FUNCTION_BLOCK FB_ReadParameterNC IMPLEMENTS I_ReadParameter
(*
    Read and refresh axis parameters
*)
VAR
    {attribute 'no_copy'}
    AxisRef : REFERENCE TO AXIS_REF;
// NC parameters that are exposed with pytmc pragmas
    {attribute 'pytmc' := '
        pv: PLC:AxisPar
        io: i
        field: DESC Axis configuration parameters in the numerical controller.
    '}
    stAxisParametersExposed : ST_AxisParameterSetExposed;

    // MC_ReadParameterSet Output
    fbMcReadParams: MC_ReadParameterSet;
    //{attribute 'hide'}
    stAxisParameters: ST_AxisParameterSet;
    bNcParamsReadInit   : BOOL;
    NCParamsTimer : TON;
    bAxisParametersInit : BOOL;
    tRefreshDelay: TIME := T#1S;
    bEnable : BOOL;
    bExecute : BOOL;
    bError				: BOOL;
    nErrorId			: UDINT:=0;
    sMessage : T_MAXSTRING;
    bDone : BOOL;
    bBusy    : BOOL;
END_VAR

PROPERTY Aborted : BOOL
GET
END_GET
END_PROPERTY

PROPERTY Active : BOOL
GET
END_GET
END_PROPERTY

PROPERTY AmsNetID : T_AmsNetId
GET
AmsNetID := THIS^.stAxisParameters.sAmsNetId;
END_GET
END_PROPERTY

PROPERTY AxisReadParamsInit : BOOL
GET
AxisReadParamsInit := bAxisParametersInit;
END_GET
END_PROPERTY

PROPERTY Busy : BOOL
GET
Busy := bBusy;
END_GET
END_PROPERTY

METHOD PUBLIC CallAfterInit
VAR_INPUT
    AxisRef : REFERENCE TO AXIS_REF;
END_VAR
THIS^.AxisRef REF= AxisRef;
END_METHOD

PROPERTY Done : BOOL
GET
Done := bDone;
END_GET
END_PROPERTY

PROPERTY EnInTargetTimeout : BOOL
GET
EnInTargetTimeout := THIS^.stAxisParameters.bEnablePEHTimeControl.0;
END_GET
END_PROPERTY

PROPERTY EnMaxSoftPosLimit : BOOL
GET
EnMaxSoftPosLimit := THIS^.stAxisParameters.bEncEnableSoftEndMaxControl.0;
END_GET
END_PROPERTY

PROPERTY EnMinSoftPosLimit : BOOL
GET
EnMinSoftPosLimit := THIS^.stAxisParameters.bEncEnableSoftEndMinControl.0;
END_GET
END_PROPERTY

PROPERTY EnPositionLagMonitoring : BOOL
GET
EnPositionLagMonitoring := THIS^.stAxisParameters.bCtrlEnablePosDiffControl.0;
END_GET
END_PROPERTY

PROPERTY EnPositionRangeMonitoring : BOOL
GET
END_GET
END_PROPERTY

PROPERTY EnScaleFactorInternal : LREAL
GET
EnScaleFactorInternal := THIS^.stAxisParameters.fEncScaleFactorInternal;
END_GET
END_PROPERTY

PROPERTY EnTargetPositionMonitoring : BOOL
GET
EnTargetPositionMonitoring := THIS^.stAxisParameters.bEnableTargetPosControl.0;
END_GET
END_PROPERTY

PROPERTY Error : BOOL
GET
Error := bError;
END_GET
END_PROPERTY

PROPERTY ErrorID : UDINT
GET
ErrorID := nErrorID;
END_GET
END_PROPERTY

//FB_Init is always available implicitly and it is used primarily for initialization.
//The return value is not evaluated. For a specific influence, you can also declare the
//methods explicitly and provide additional code there with the standard initialization
//code. You can evaluate the return value.
METHOD FB_Init: BOOL
VAR_INPUT
    bInitRetains: BOOL; // TRUE: the retain variables are initialized (reset warm / reset cold)
    bInCopyCode: BOOL;  // TRUE: the instance will be copied to the copy code afterward (online change)
    AxisRef : REFERENCE TO AXIS_REF;
END_VAR
THIS^.AxisRef REF= AxisRef;
END_METHOD

PROPERTY InTargetTimeout : LREAL
GET
InTargetTimeout := THIS^.stAxisParameters.fPEHControlTime;
END_GET
END_PROPERTY

PROPERTY MaxPosLagFilterTime : LREAL
GET
MaxPosLagFilterTime := THIS^.stAxisParameters.fCtrlPosDiffMaxTime;
END_GET
END_PROPERTY

PROPERTY MaxPosLagValue : LREAL
GET
MaxPosLagValue := THIS^.stAxisParameters.fCtrlPosDiffMax;
END_GET
END_PROPERTY

PROPERTY MaxSoftPosLimit : LREAL
GET
MaxSoftPosLimit := THIS^.stAxisParameters.fEncSoftEndMax;
END_GET
END_PROPERTY

PROPERTY Message : T_MAXSTRING
GET
Message := sMessage;
END_GET
END_PROPERTY

PROPERTY MinSoftPosLimit : LREAL
GET
MinSoftPosLimit := THIS^.stAxisParameters.fEncSoftEndMin;
END_GET
END_PROPERTY

PROPERTY Port : WORD
GET
Port := THIS^.stAxisParameters.nPort;
END_GET
END_PROPERTY

PROPERTY PositionRangeWindow : LREAL
GET
END_GET
END_PROPERTY

METHOD ReadParameters
VAR_INPUT
    Enable: BOOL;
    RefreshDelay: TIME;
END_VAR
THIS^.bEnable:= Enable;
THIS^.tRefreshDelay:= RefreshDelay;
END_METHOD

PROPERTY RefVeloSearch : LREAL
GET
RefVeloSearch := THIS^.stAxisParameters.fRefVeloSearch;
END_GET
END_PROPERTY

PROPERTY RefVeloSync : LREAL
GET
RefVeloSync:= THIS^.stAxisParameters.fRefVeloSync;
END_GET
END_PROPERTY

PROPERTY TargetPositionMonitoringTime : LREAL
GET
TargetPositionMonitoringTime := THIS^.stAxisParameters.fTargetPosControlTime;
END_GET
END_PROPERTY

PROPERTY TargetPositionWindow : LREAL
GET
TargetPositionWindow := THIS^.stAxisParameters.fTargetPosControlRange;
END_GET
END_PROPERTY

END_FUNCTION_BLOCK

(* stored: Version 1.1.0.1
   POU FB_ReadParameterNC: Id {0a080461-8875-4b57-a673-44abaad03a9d}, SpecialFunc None
   Property Aborted: Id {eb6c713a-ae14-4aae-8e2a-0fe4445d0481}
   Get Get: Id {f67f949f-e2ba-4069-927a-e0e24cc413f2}
   Property Active: Id {801f778e-5bb2-47d5-80a0-c3ed9d0e6e0e}
   Get Get: Id {55e2ced6-d12a-441b-af90-d38eb2a717d3}
   Property AmsNetID: Id {79cec594-74b3-4c58-9634-32ff2e3930e8}
   Get Get: Id {26a88863-17bb-47a9-a2bd-19cbf4755392}
   Property AxisReadParamsInit: Id {78f88bc3-cc72-458c-8f2d-1ca8c5361c73}
   Get Get: Id {c9c8de24-42ba-4328-8718-b4ef40ba79c8}
   Property Busy: Id {22f692ee-01c6-4a60-890c-87d05d869350}
   Get Get: Id {cb5a710f-fdfd-425d-a3db-4a2ca84d2713}
   Method CallAfterInit: Id {f18b7d6f-c3da-460b-84aa-32d432fd132a}
   Property Done: Id {6a425195-42c1-4362-9605-a1abf17cb028}
   Get Get: Id {a7bf1f50-dd9e-4d56-8de5-d617db746ffc}
   Property EnInTargetTimeout: Id {cb614f62-92c0-4ff8-b236-945144e388d5}
   Get Get: Id {e76567d5-05fc-4d20-b5e3-13501c35b76c}
   Property EnMaxSoftPosLimit: Id {3c3b7f0e-0e4c-4285-8283-374d54e7aebe}
   Get Get: Id {5bf87a4b-90bb-42bd-aa83-7f5af523ba2e}
   Property EnMinSoftPosLimit: Id {bb2ca3a8-8fc7-44bd-bb8b-f57f80462214}
   Get Get: Id {2bde1d8a-8373-4f56-af76-c94a528845e6}
   Property EnPositionLagMonitoring: Id {29f614c8-318b-43a9-8822-edab8f52e92e}
   Get Get: Id {a531602a-dfcd-412c-be97-8fd45db94be1}
   Property EnPositionRangeMonitoring: Id {f8605e66-e221-4fcd-9b0f-84d9ba4e2637}
   Get Get: Id {57d74d2c-0ebe-4765-965f-ec15ea6e2adc}
   Property EnScaleFactorInternal: Id {96b925d2-167e-491a-8875-bd75d9890a67}
   Get Get: Id {0b20ae66-5839-48f1-b958-6e8d6608e6e3}
   Property EnTargetPositionMonitoring: Id {3579721b-0625-4781-83f8-4617310d0f0c}
   Get Get: Id {06fd4c5e-7b2b-4004-898a-fbf20b3937b1}
   Property Error: Id {9c9b784c-64ad-45f6-9c7e-0135e01c740f}
   Get Get: Id {81197bc9-252b-4651-b7ec-0e59bda13a17}
   Property ErrorID: Id {54050bbe-c894-4265-8ce6-db4f8c907c4e}
   Get Get: Id {51259382-0371-44cd-8353-1addb15d13a4}
   Method FB_Init: Id {9a2f321a-6442-4481-94f8-cad0f90b6a8f}
   Property InTargetTimeout: Id {3f12d2a6-41fc-4962-a67a-6325c2241f2e}
   Get Get: Id {9e1e4a5e-97db-4ea8-9aca-15c2d5b81320}
   Property MaxPosLagFilterTime: Id {1feeb96a-18f8-4ecf-9c69-fb4f8bfd7dbe}
   Get Get: Id {64ba684b-07d9-4327-9788-034ad75501f1}
   Property MaxPosLagValue: Id {843bf621-4ed1-478c-9c6c-f985742062a8}
   Get Get: Id {8a9ca48f-156e-4613-87a3-f910f9ec0e0b}
   Property MaxSoftPosLimit: Id {7744fb96-6717-48b6-a170-01beef3e12c1}
   Get Get: Id {8efc13a2-8787-4a6f-af46-e11f1d25d992}
   Property Message: Id {5a724cf4-bb87-4860-9c8b-1548832af991}
   Get Get: Id {0e6a7eb8-6fa2-4ab3-ba2f-5e01d94ba75a}
   Property MinSoftPosLimit: Id {ae44b4d0-7941-4537-a170-677565224641}
   Get Get: Id {a1d48c0a-3f6a-4cab-b8e6-43da7538de47}
   Property Port: Id {c338a91a-3ae5-4a47-941b-0449f157640f}
   Get Get: Id {9af1eadb-d648-4a5e-8241-ff6553a4a709}
   Property PositionRangeWindow: Id {1dd8cb74-3cd9-4b43-9ddb-21cd3c83088d}
   Get Get: Id {e182bb73-32dd-43f1-baa8-64f5fd1417df}
   Method ReadParameters: Id {7e1988df-13bf-409f-9bba-5c8975b3fe8b}
   Property RefVeloSearch: Id {8705c180-d9e3-4f14-a09b-5c1fee343bd9}
   Get Get: Id {cc5c8632-aa63-4a37-8470-a4ffc3f9a6d9}
   Property RefVeloSync: Id {c30dca5c-0998-42d3-aa48-35c4d73ce582}
   Get Get: Id {700b38d3-f6d3-4d02-a47e-cfd3c1cbbb52}
   Property TargetPositionMonitoringTime: Id {e3fcf39b-d48d-452b-acdd-8281cb10837a}
   Get Get: Id {a626b81c-5dfd-4cab-adb5-aa6cb8402380}
   Property TargetPositionWindow: Id {0f7050ba-57af-4a1f-8073-9d5358da6478}
   Get Get: Id {61318993-34b7-4456-9141-97cc30829e83} *)
